(* CoDeSys 2.3.9.50 project: 8A.pr6 *)
(* Libraries: STANDARD.LB6 5.6.98 12:03:02 *)

(* POU MAIN, LD *)
PROGRAM MAIN
VAR
	Fully_closed AT %IX0.0: BOOL;
	Fully_opened AT %IX0.1: BOOL;
	UP AT %IX0.2: BOOL;
	DOWN AT %IX0.3: BOOL;
	Stop AT %IX0.4: BOOL;
	UP_Light AT %QX0.0: BOOL;
	DOWN_Light AT %QX0.1: BOOL;
	Current: INT := 0;
	final: INT;
	reset AT %IX7.7: BOOL;
	Opened AT %QX0.3: BOOL;
	Closed AT %QX0.2: BOOL;
	Partially_open AT %QX0.5: BOOL;
	Red_light AT %QX0.6: BOOL;
	Green_Light AT %QX0.7: BOOL;
	yellow_Light AT %QX1.0: BOOL;
	Forward_motor AT %QX1.1: BOOL;
	Reversed_motor AT %QX1.2: BOOL;
END_VAR
VAR (* helpers for the ST form of the networks *)
	_p1 : BOOL;
	_p2 : BOOL;
END_VAR
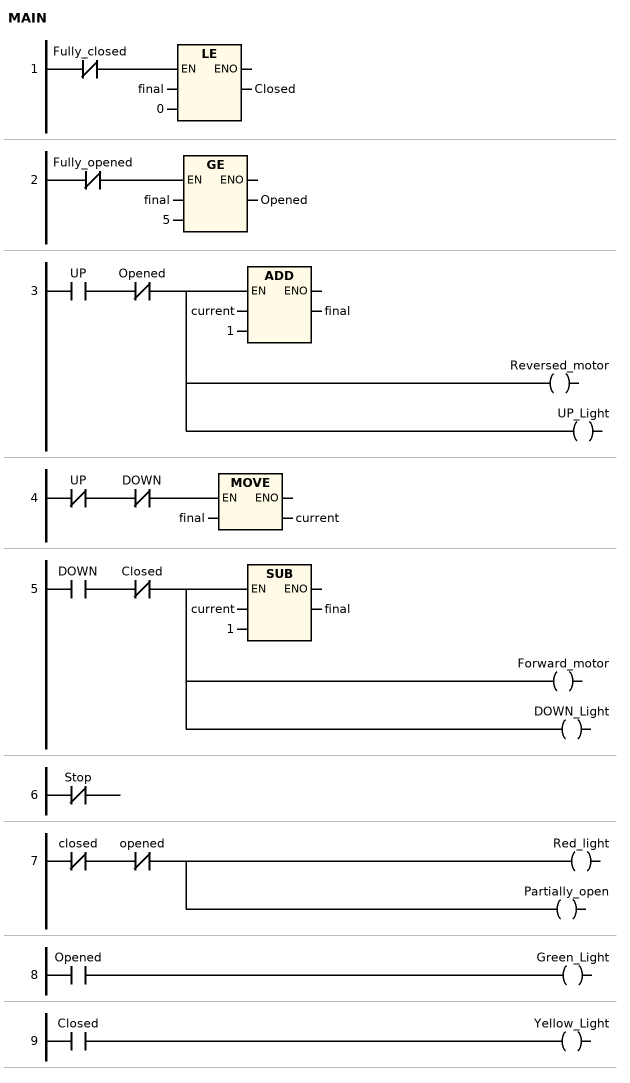
_LD_ (* Ladder Diagram *)
NETWORK 1
	[/Fully_closed]
		EN --- LE(final, 0) => Closed
NETWORK 2
	[/Fully_opened]
		EN --- GE(final, 5) => Opened
NETWORK 3
	[UP] - [/Opened] --- (Reversed_motor) (UP_Light)
		EN --- ADD(current, 1) => final
NETWORK 4
	[/UP] - [/DOWN]
		EN --- MOVE(final) => current
NETWORK 5
	[DOWN] - [/Closed] --- (Forward_motor) (DOWN_Light)
		EN --- SUB(current, 1) => final
NETWORK 6
	[/Stop]
NETWORK 7
	[/closed] - [/opened] --- (Red_light) (Partially_open)
NETWORK 8
	[Opened] --- (Green_Light)
NETWORK 9
	[Closed] --- (Yellow_Light)
_END_LD_
(* the same logic as Structured Text *)
(* Network 1 *)
IF NOT Fully_closed THEN
	Closed := final <= 0;
END_IF;
(* Network 2 *)
IF NOT Fully_opened THEN
	Opened := final >= 5;
END_IF;
(* Network 3 *)
_p1 := UP AND NOT Opened;
IF _p1 THEN
	final := current + 1;
END_IF;
Reversed_motor := _p1;
UP_Light := _p1;
(* Network 4 *)
IF NOT UP AND NOT DOWN THEN
	current := final;
END_IF;
(* Network 5 *)
_p2 := DOWN AND NOT Closed;
IF _p2 THEN
	final := current - 1;
END_IF;
Forward_motor := _p2;
DOWN_Light := _p2;
(* Network 6 *)
(* Network 7 *)
Red_light := NOT closed AND NOT opened;
Partially_open := Red_light;
(* Network 8 *)
Green_Light := Opened;
(* Network 9 *)
Yellow_Light := Closed;
END_PROGRAM
